// LS Electric XG5000 project: 14_전등제어
// PLC NewPLC
// module base 0 slot 0: 입출력 모듈:XBC-DN/DP14E (DC 24V 입력 8점, 트랜지스터 출력 6점)

PROGRAM NewProgram (task: 스캔 프로그램)

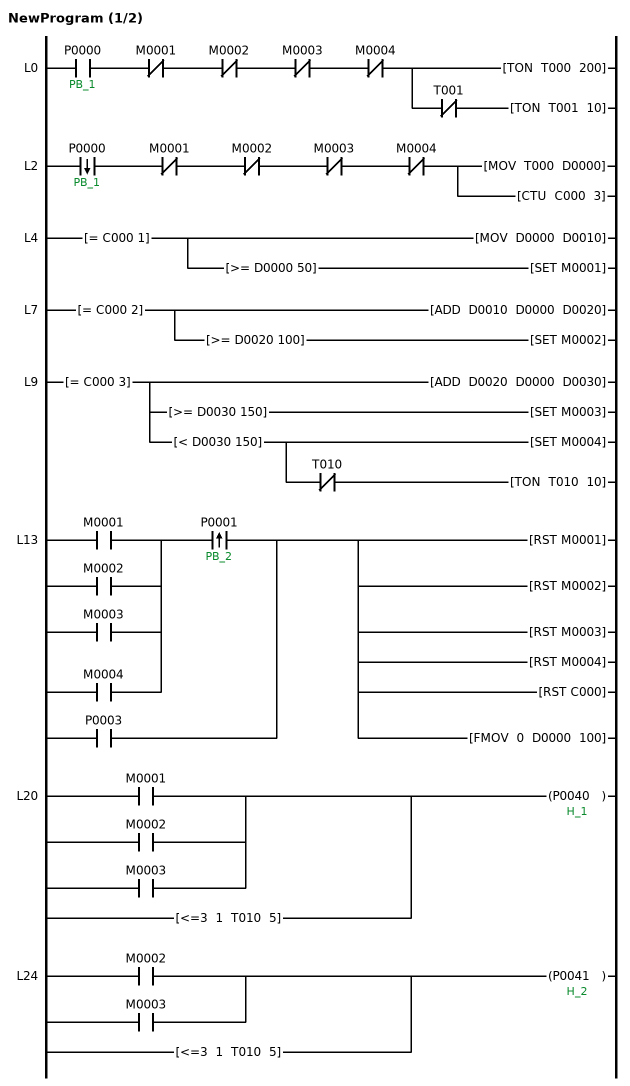
; L0
LOAD      P0000	// PB_1
AND NOT   M0001
AND NOT   M0002
AND NOT   M0003
AND NOT   M0004
TON       T000 200
AND NOT   T001
TON       T001 10
; L2
LOADN     P0000	// PB_1
AND NOT   M0001
AND NOT   M0002
AND NOT   M0003
AND NOT   M0004
MOV       T000 D0000
CTU       C000 3
; L4
LOAD=     C000 1
MOV       D0000 D0010
AND>=     D0000 50
SET       M0001
; L7
LOAD=     C000 2
ADD       D0010 D0000 D0020
AND>=     D0020 100
SET       M0002
; L9
LOAD=     C000 3
ADD       D0020 D0000 D0030
MPUSH
AND>=     D0030 150
SET       M0003
MPOP
AND<      D0030 150
SET       M0004
AND NOT   T010
TON       T010 10
; L13
LOAD      M0001
OR        M0002
OR        M0003
OR        M0004
ANDP      P0001	// PB_2
OR        P0003
RST       M0001
RST       M0002
RST       M0003
RST       M0004
RST       C000
FMOV      0 D0000 100
; L20
LOAD      M0001
OR        M0002
OR        M0003
OR<=3     1 T010 5
OUT       P0040	// H_1
; L24
LOAD      M0002
OR        M0003
OR<=3     1 T010 5
OUT       P0041	// H_2

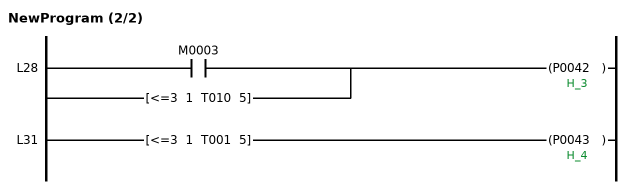
; L28
LOAD      M0003
OR<=3     1 T010 5
OUT       P0042	// H_3
; L31
LOAD<=3   1 T001 5
OUT       P0043	// H_4